(* Logix 5000 project; controller NorthLineDepalletizerPLC vendor 1 type 14 code 106 rev 33.11; software revision 33.00 *)

TASK MainTask (continuous, watchdog 500 ms) : MainProgram, Motoman, Comms

MODULES
   Local : vendor 1 type 14 code 106 (Compact 0, rev 33.11)
      BrazingOvenEthernetCard : 1756-ENBT (Ethernet 192.168.1.100, rev 5.1, Output RPI 10 ms)
         BrazingOvenPLC : vendor 1 type 14 code 92 (ICP 0, rev 24.1, $af6df9d4$ RPI 20 ms)
      cam : vendor 678 type 100 code 276 (Ethernet 192.168.1.33, rev 11.1, Output RPI 60 ms)
      YRC1000_Rbt_Ctlr : ETHERNET-MODULE (Ethernet 192.168.1.31, rev 1.1, Output RPI 10 ms)
      Fanuc_5 : ETHERNET-MODULE (Ethernet 192.168.1.5, rev 1.1, Output RPI 10 ms)
           Fanuc_5:I.Data[2]   // Part Count from Fanuc
           Fanuc_5:O.Data[0]   // Part Width to give to Fanuc
           Fanuc_5:O.Data[3]   // Part Length to give to Fanuc
           Fanuc_5:O.Data[1]   // Part ID to give to Fanuc
           Fanuc_5:O.Data[4]   // Part Count to give to Fanuc
           Fanuc_5:O.Data[2]   // Conveyor Height to pass along to Fanuc
      IFM_AL1322 : vendor 322 type 12 code 1322 (Ethernet 192.168.1.32, rev 1.6, StandardDataDriven RPI 10 ms)
END_MODULES

TYPE PatternResult :
STRUCT
   Angle : REAL;
   Score : REAL;
   X : REAL;
   Y : REAL;
END_STRUCT
END_TYPE

TYPE YRC1000_POSITION_VAR :
STRUCT
   Data_Type : DINT;   // Position Data Type of the Following Data 0: Pulse 16: Base 17: Robot 18: Tool 19: User coordinates
   Config : DINT;   // The configuration will be output bit 0: Back bit 1: Lower arm bit 2: No flip bit 3: R axis ≥ 180° bit 4: T axis ≥ 180° bit 5: S axis ≥ 180°
   Tool_Num : DINT;   // Tool #
   User_Coord_Num : DINT;   // User Coordinate #
   Ext_Config : DINT;   // Output the 7-axis robot extended configuration bit 0: θL ≥ 180° bit 1: θU ≥ 180° bit 2: θB ≥ 180° bit 3: θE ≥ 180° bit 4: θW ≥ 180°
   Axis1_Data : DINT;   // For pulse: Each axis’ pulse value For base: Length (μm) Angle (0.0001°)
   Axis2_Data : DINT;   // For pulse: Each axis’ pulse value For base: Length (μm) Angle (0.0001°)
   Axis3_Data : DINT;   // For pulse: Each axis’ pulse value For base: Length (μm) Angle (0.0001°)
   Axis4_Data : DINT;   // For pulse: Each axis’ pulse value For base: Length (μm) Angle (0.0001°)
   Axis5_Data : DINT;   // For pulse: Each axis’ pulse value For base: Length (μm) Angle (0.0001°)
   Axis6_Data : DINT;   // For pulse: Each axis’ pulse value For base: Length (μm) Angle (0.0001°)
   Axis7_Data : DINT;   // For pulse: Each axis’ pulse value For base: Length (μm) Angle (0.0001°)
   Axis8_Data : DINT;   // For pulse: Each axis’ pulse value For base: Length (μm) Angle (0.0001°)
END_STRUCT
END_TYPE

ADD_ON_INSTRUCTION Generic_8PORT_IOL   (* revision 3.0 *)
// Revision note:
// 12/2022:updated to current AOI standards:LH
VAR_IN_OUT
   PLC_Input : INT[223]; {required}   // Reference the Input Controller tag <IOLinkMasterName>:I1.Data
   PLC_Output : INT[151]; {required}   // Reference the Output Controller tag <IOLinkMasterName>:O1.Data
END_VAR
VAR_INPUT
   Port_Process_Data_Size : SINT := 4;   // User Input Value from the Configuration Controller tag <IOLinkMasterName>:C.Port_Process_Data_Size
   Port_Number : SINT; {visible}   // User Input Value = Port number of the IO-Link Master
END_VAR
VAR_OUTPUT
   Vendor_ID : INT; {access Read Only, visible}   // Read only value indicating the manufacturer of the IO-Link Device. ifm=310 dec
   Device_ID : DINT; {access Read Only, visible}   // Read only value set by the manufacturer of the device. Varies by product family
   IOL_Mode : BOOL; {access Read Only, visible}   // True: Port is configured for IO-Link Communication. False: Port is not configured for IO-Link Communication
   Device_Not_Connected : BOOL; {access Read Only, visible}   // True: No IO-Link Device is connected False: IO-Link Device is connected
   Invalid_Data : BOOL; {access Read Only, visible}   // True: IO-Link Data is invalid False: IO-Link Data is valid
   Wrong_VID_DID : BOOL; {access Read Only, visible}   // True: Vendor ID and/or Device ID does not match the configured VID or DID set in Configuration Controller Tag(s) <IOLink MasterName>:C.Vendor_ID_Port_n or ...C.Device_ID_Port_n
   Diagnostic_Avail : BOOL; {access Read Only, visible}   // True: IO-Link Event data is available False: No Event data is present
   AOI_Settings_Error : BOOL; {access Read Only, visible}   // A user input is out of range. Check port process data size and port number
END_VAR
VAR_IN_OUT
   Input_Data_Array : INT[16]; {required}   // Up to 16 words/32 bytes of Input process data produced by the IO-Link device
        [5]   // Input Word 5/Byte 10 0..7/Byte 11 8..15
        [0]   // Input Word 0/Byte 0 0..7/Byte 1 8..15
        [1]   // Input Word 1/Byte 2 0..7/Byte 3 8..15
        [6]   // Input Word 6/Byte 12 0..7/Byte 13 8..15
        [2]   // Input Word 2/Byte 4 0..7/Byte 5 8..15
        [7]   // Input Word 7/Byte 14 0..7/Byte 15 8..15
        [8]   // Input Word 8/Byte 16 0..7/Byte 17 8..15
        [9]   // Input Word 9/Byte 18 0..7/Byte 19 8..15
        [3]   // Input Word 3/Byte 6 0..7/Byte 7 8..15
        [10]   // Input Word 10/Byte 20 0..7/Byte 21 8..15
        [11]   // Input Word 11/Byte 22 0..7/Byte 23 8..15
        [12]   // Input Word 12/Byte 24 0..7/Byte 25 8..15
        [13]   // Input Word 13/Byte 26 0..7/Byte 27 8..15
        [14]   // Input Word 14/Byte 28 0..7/Byte 29 8..15
        [15]   // Input Word 15/Byte 30 0..7/Byte 31 8..15
        [4]   // Input Word 4/Byte 8 0..7/Byte 9 8..15
   Output_Data_Array : INT[16]; {required}   // Up to 32 bytes of Output process data consumed by the IO-Link device
        [0]   // Output Word 0/Byte 1 0..7/Byte 0 8..15
        [1]   // Output Word 1/Byte 3 0..7/Byte 2 8..15
        [5]   // Output Word 5/Byte 11 0..7/Byte 10 8..15
        [6]   // Output Word 6/Byte 13 0..7/Byte 12 8..15
        [7]   // Output Word 7/Byte 15 0..7/Byte 14 8..15
        [8]   // Output Word 8/Byte 17 0..7/Byte 16 8..15
        [9]   // Output Word 9/Byte 19 0..7/Byte 18 8..15
        [2]   // Output Word 2/Byte 5 0..7/Byte 4 8..15
        [3]   // Output Word 3/Byte 7 0..7/Byte 6 8..15
        [10]   // Output Word 10/Byte 21 0..7/Byte 20 8..15
        [4]   // Output Word 4/Byte 9 0..7/Byte 8 8..15
        [11]   // Output Word 11/Byte 23 0..7/Byte 22 8..15
        [12]   // Output Word 12/Byte 25 0..7/Byte 24 8..15
        [13]   // Output Word 13/Byte 27 0..7/Byte 26 8..15
        [14]   // Output Word 14/Byte 29 0..7/Byte 28 8..15
        [15]   // Output Word 15/Byte 31 0..7/Byte 30 8..15
END_VAR
VAR
   Data_Size : SINT; {access None}   // Factor of the RealPort_Num to calcualated the Offset_Address
   Offset_StatusFlgs : SINT; {access None}   // RealPort_Num+9
   RealPort_Num : SINT; {access None}   // Result of the Port_Number-1
   StatusFlgs_Offset : SINT; {access None}   // Result of Offset_StatusFlgs+23
   Offset_Address : INT; {access None}   // Result of Data_Size*RealPort_Number
   Process_Offset : INT; {access None}   // Result of Offset_Address+95(8port Master) or Offset_Address+59(4port Master). Used to indicate the word offset for where the IO-Link device’s process input data starts
   Process_Out_Offset : INT; {access None}   // Result of Offset_Address+23
END_VAR

ROUTINE Logic   (* ladder *)
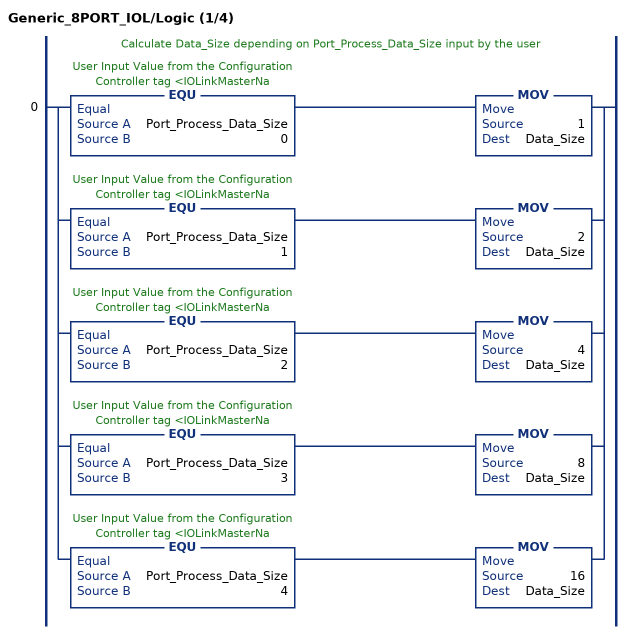
   // Calculate Data_Size depending on Port_Process_Data_Size input by the user
   0: [EQU(Port_Process_Data_Size,0) MOV(1,Data_Size) ,EQU(Port_Process_Data_Size,1) MOV(2,Data_Size) ,EQU(Port_Process_Data_Size,2) MOV(4,Data_Size) ,EQU(Port_Process_Data_Size,3) MOV(8,Data_Size) ,EQU(Port_Process_Data_Size,4) MOV(16,Data_Size) ];
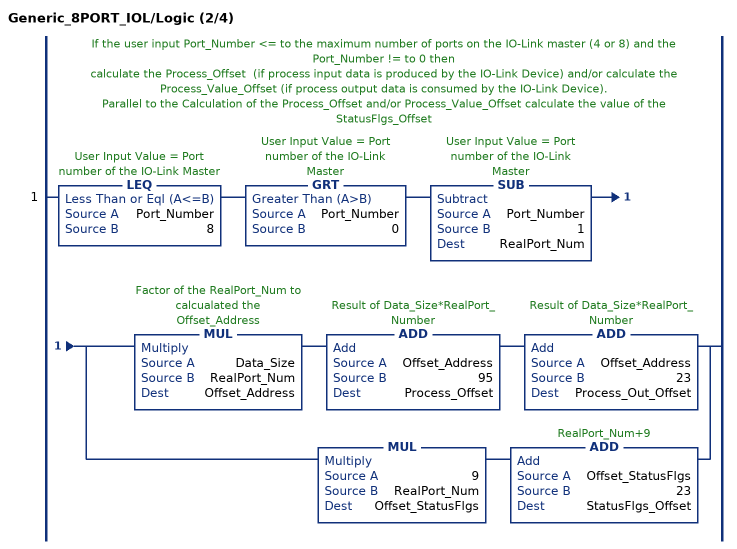
   // If the user input Port_Number <= to the maximum number of ports on the IO-Link master (4 or 8) and the Port_Number != to 0 then
   // calculate the Process_Offset  (if process input data is produced by the IO-Link Device) and/or calculate the Process_Value_Offset (if process output data is consumed by the IO-Link Device).
   // Parallel to the Calculation of the Process_Offset and/or Process_Value_Offset calculate the value of the StatusFlgs_Offset
   1: LEQ(Port_Number,8)GRT(Port_Number,0)SUB(Port_Number,1,RealPort_Num)[MUL(Data_Size,RealPort_Num,Offset_Address) ADD(Offset_Address,95,Process_Offset) ADD(Offset_Address,23,Process_Out_Offset) ,MUL(9,RealPort_Num,Offset_StatusFlgs) ADD(Offset_StatusFlgs,23,StatusFlgs_Offset) ];
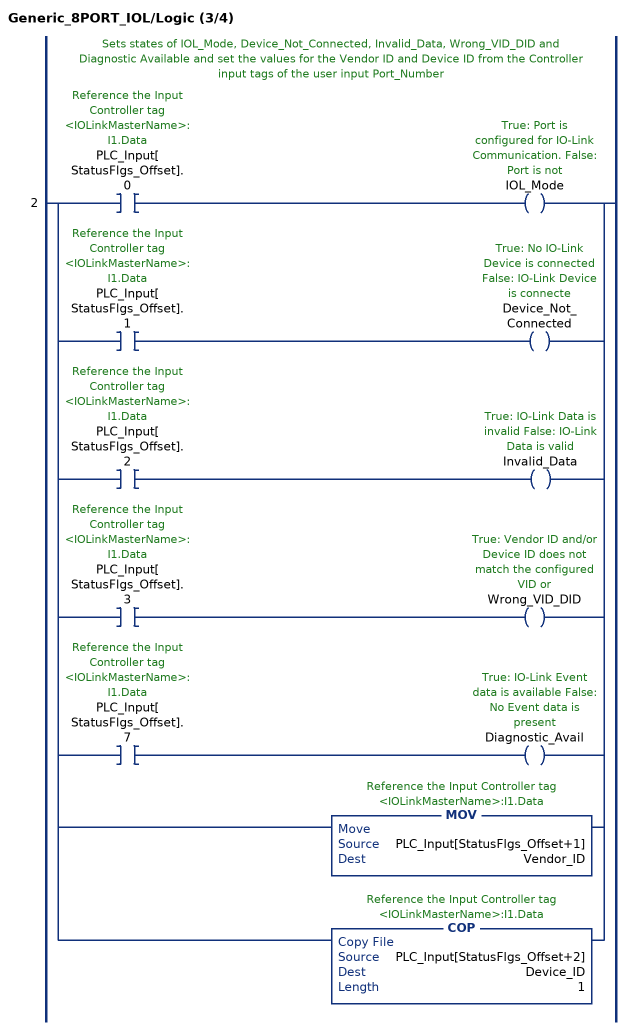
   // Sets states of IOL_Mode, Device_Not_Connected, Invalid_Data, Wrong_VID_DID and Diagnostic Available and set the values for the Vendor ID and Device ID from the Controller input tags of the user input Port_Number
   2: [XIC(PLC_Input[StatusFlgs_Offset].0) OTE(IOL_Mode) ,XIC(PLC_Input[StatusFlgs_Offset].1) OTE(Device_Not_Connected) ,XIC(PLC_Input[StatusFlgs_Offset].2) OTE(Invalid_Data) ,XIC(PLC_Input[StatusFlgs_Offset].3) OTE(Wrong_VID_DID) ,XIC(PLC_Input[StatusFlgs_Offset].7) OTE(Diagnostic_Avail) ,MOV(PLC_Input[StatusFlgs_Offset+1],Vendor_ID) ,COP(PLC_Input[StatusFlgs_Offset+2],Device_ID,1) ];
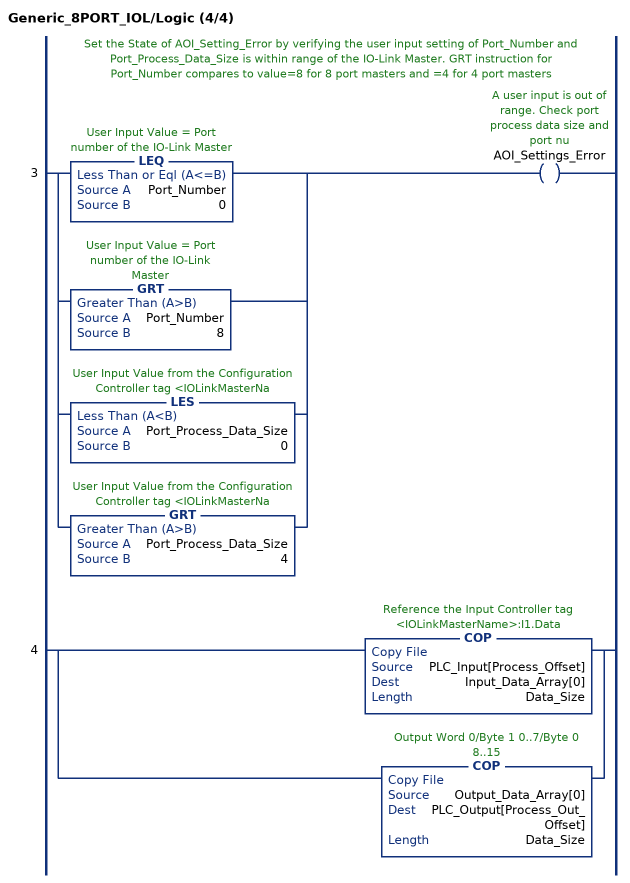
   // Set the State of AOI_Setting_Error by verifying the user input setting of Port_Number and Port_Process_Data_Size is within range of the IO-Link Master. GRT instruction for Port_Number compares to value=8 for 8 port masters and =4 for 4 port masters
   3: [LEQ(Port_Number,0) ,GRT(Port_Number,8) ,LES(Port_Process_Data_Size,0) ,GRT(Port_Process_Data_Size,4) ]OTE(AOI_Settings_Error);
   4: [COP(PLC_Input[Process_Offset],Input_Data_Array[0],Data_Size) ,COP(Output_Data_Array[0],PLC_Output[Process_Out_Offset],Data_Size) ];
END_ROUTINE
END_ADD_ON_INSTRUCTION

VAR_GLOBAL   (* controller tags *)
   AcknowledgeCameraImage : ALIAS FOR YRC1000_Rbt_Ctlr:O.Data[4].5;
   AcknowledgeHeightCheck : ALIAS FOR YRC1000_Rbt_Ctlr:O.Data[4].4;
   AcknowledgeLevelCheck : ALIAS FOR YRC1000_Rbt_Ctlr:O.Data[6].4;
   AcknowledgePalletTooTall : ALIAS FOR YRC1000_Rbt_Ctlr:O.Data[7].4;
   ActiveUserFrame : DINT;   // Currently Active Pallet
   AirPressure : ALIAS FOR YRC1000_Rbt_Ctlr:I.Data[1].4;
   Alarm : ALIAS FOR YRC1000_Rbt_Ctlr:I.Data[8].3;
   AlarmReset : ALIAS FOR YRC1000_Rbt_Ctlr:O.Data[0].3;
   AngleHeightCheck : ALIAS FOR YRC1000_Rbt_Ctlr:I.Data[10].4;
   AtHomePosition : ALIAS FOR YRC1000_Rbt_Ctlr:I.Data[5].2;
   BatteryAlarm : ALIAS FOR YRC1000_Rbt_Ctlr:I.Data[8].4;
   Blue1 : BOOL;
   Blue2 : BOOL;
   CallMaster : ALIAS FOR YRC1000_Rbt_Ctlr:O.Data[0].2;
   CameraAngle : REAL := 0.56835175;
   CameraFailed : ALIAS FOR YRC1000_Rbt_Ctlr:O.Data[5].7;
   CameraJobName : STRING := '2832_SingleStackACoils.job';
   CameraOffsetX : REAL := 0.8950585;
   CameraOffsetY : REAL := -5.923684;
   CameraScore : REAL := 1.0;
   CamJobData : SINT[32] := ([0] := 26, [2] := 50, [3] := 56, [4] := 51, [5] := 50, [6] := 95, [7] := 83, [8] := 105, [9] := 110, [10] := 103, [11] := 108, [12] := 101, [13] := 83, [14] := 116, [15] := 97, [16] := 99, [17] := 107, [18] := 65, [19] := 67, [20] := 111, [21] := 105, [22] := 108, [23] := 115, [24] := 46, [25] := 106, [26] := 111, [27] := 98);
   CapacitiveInArray : INT[16] := ([0] := 928);
   CapacitiveOutArray : INT[16];
   CapacitiveSensorValue : DINT := 58;
   ccr0 : DINT;
   ccr1 : DINT := 1;
   ccr2 : DINT := 2;
   ChangingJob : BOOL;
   CoilLocation : YRC1000_POSITION_VAR := (Data_Type := 19, Tool_Num := 2, User_Coord_Num := 5, Axis1_Data := 895, Axis2_Data := -5924, Axis3_Data := 15000, Axis4_Data := 1800000, Axis6_Data := -1794316);
   CoilLocationFound : ALIAS FOR YRC1000_Rbt_Ctlr:O.Data[4].6;
   CoilType : DINT := 1;   // 1: 17" 2: 30" 3: 41"
   CompleteState : DINT := 100;
   ConvertedCameraResults : REAL[3] := ([0] := 0.8950585, [1] := -5.923684, [2] := -179.43164);
   ConveyorApproach : YRC1000_POSITION_VAR := (Data_Type := 19, Tool_Num := 8, User_Coord_Num := 3, Axis2_Data := -50000, Axis3_Data := 151600, Axis4_Data := 1800000, Axis5_Data := 100000, Axis6_Data := -900000);
   ConveyorBeforePlace : YRC1000_POSITION_VAR := (Data_Type := 19, Tool_Num := 8, User_Coord_Num := 3, Axis2_Data := -10000, Axis3_Data := 56600, Axis4_Data := 1800000, Axis5_Data := 100000, Axis6_Data := -900000);
   ConveyorIn : YRC1000_POSITION_VAR := (Data_Type := 19, Tool_Num := 8, User_Coord_Num := 3, Axis2_Data := -50000, Axis3_Data := 56600, Axis4_Data := 1800000, Axis5_Data := 100000, Axis6_Data := -900000);
   ConveyorOver : YRC1000_POSITION_VAR := (Data_Type := 19, Tool_Num := 8, User_Coord_Num := 3, Axis2_Data := -50000, Axis3_Data := 151600, Axis4_Data := 1800000, Axis5_Data := 100000, Axis6_Data := -900000);
   Corner1Dist : DINT := 1499300;
   Corner2Dist : DINT := 1508800;
   Corner3Dist : DINT := 1504500;
   Corner4Dist : DINT := 1504900;
   Cos30 : REAL := 0.8660254;
   Cos45 : REAL := 0.70710677;
   CurrentPos : REAL[6] := ([0] := 1000.0, [2] := 799.997, [3] := 180.0, [4] := -0.0003, [5] := -1.e-04);   // Current position of the active TCP on the robot
   CurrentPosition_micro : YRC1000_POSITION_VAR := (Data_Type := 16, Config := 4, Tool_Num := 1, Axis1_Data := 1000000, Axis3_Data := 799997, Axis4_Data := 1800000, Axis5_Data := -3, Axis6_Data := -1);
   CurrentRobotTask : DINT := 5;
   delay_0017_Coil_Camera : TIMER := (PRE := 10);
   delay_0017_Orient_Camera : TIMER := (PRE := 10);
   delay_0017_PickLocation : TIMER := (PRE := 10, ACC := 10, EN := 1, DN := 1);
   delay_2832_Edge_Camera : TIMER := (PRE := 10);
   delay_2832_Edge_SearchLocation : TIMER := (PRE := 10);
   delay_2832_Middle_Camera : TIMER := (PRE := 10);
   delay_2832_Middle_SearchLocation : TIMER := (PRE := 10);
   delay_2832_PickLocation : TIMER := (PRE := 10);
   delay_3041_Edge_Camera : TIMER := (PRE := 10);
   delay_3041_Edge_SearchLocation : TIMER := (PRE := 10);
   delay_3041_Middle_Camera : TIMER := (PRE := 10);
   delay_3041_Middle_SearchLocation : TIMER := (PRE := 10, ACC := 11, EN := 1, DN := 1);
   delay_3041_PickLocation : TIMER := (PRE := 10, ACC := 11, EN := 1, DN := 1);
   delay_ActiveUserFrame : TIMER := (PRE := 10);
   delay_CurrentPos : TIMER := (PRE := 10);
   delay_LeftConveyorOff : TIMER := (PRE := 1000, ACC := 1000, EN := 1, DN := 1);
   delay_LeftConveyorOffLong : TIMER := (PRE := 60000);
   delay_LeftConveyorOn : TIMER := (PRE := 10);
   delay_LeftPalletOff : TIMER := (PRE := 1000);
   delay_LeftPalletOn : TIMER := (PRE := 1000, ACC := 1000, EN := 1, DN := 1);
   delay_PalletComplete : TIMER := (PRE := 10, ACC := 11, EN := 1, DN := 1);
   delay_Read_PartCount : TIMER := (PRE := 50, ACC := 4, EN := 1, TT := 1);
   delay_Read_RobotCurrentTask : TIMER := (PRE := 50, ACC := 38, EN := 1, TT := 1);
   delay_RightConveyorOff : TIMER := (PRE := 1000);
   delay_RightConveyorOffLong : TIMER := (PRE := 60000);
   delay_RightConveyorOn : TIMER := (PRE := 10, ACC := 10, EN := 1, DN := 1);
   delay_RightPalletOff : TIMER := (PRE := 1000, ACC := 1000, EN := 1, DN := 1);
   delay_RightPalletOn : TIMER := (PRE := 1000);
   DiffHeightCheckVal : DINT := 9500;   // Difference between the highest and shortest corners of a pallet
   DistanceInArray : INT[16] := ([0] := 22177);
        [0]   // Distance sensor reading in 0.1 mm
   DistanceOutArray : INT[16];
   DistanceSensorValue_micro : DINT := 2217600;
   DoorEntryRequested : ALIAS FOR YRC1000_Rbt_Ctlr:O.Data[5].3;
   DoorLatchRelayPower : ALIAS FOR YRC1000_Rbt_Ctlr:O.Data[2].3;
   DoorRequestAccess : ALIAS FOR YRC1000_Rbt_Ctlr:I.Data[1].0;
   DoorUnlocked : ALIAS FOR YRC1000_Rbt_Ctlr:I.Data[1].7;
   err_CameraFailed : BOOL;
   err_HeightCheckInconsistent : ALIAS FOR YRC1000_Rbt_Ctlr:O.Data[6].3;
   err_RobotPickupFailed : ALIAS FOR YRC1000_Rbt_Ctlr:I.Data[10].3;
   ErrorState : DINT := 99;
   ExternalHold : ALIAS FOR YRC1000_Rbt_Ctlr:O.Data[0].1;
   ExternalServoOn : ALIAS FOR YRC1000_Rbt_Ctlr:O.Data[0].4;
   ExternalStart : ALIAS FOR YRC1000_Rbt_Ctlr:O.Data[0].0;
   FailedCaptures : DINT;   // Number of times the camera failed to find the coil
   FanucLongPart : DINT := 1072;
   FanucMediumPart : DINT := 795;
   FanucShortPart : DINT := 465;
   FoundPattern : DINT;
   GoHome : ALIAS FOR YRC1000_Rbt_Ctlr:O.Data[6].6;
   GoodToPick : ALIAS FOR YRC1000_Rbt_Ctlr:O.Data[8].0;
   GoToToolChange : ALIAS FOR YRC1000_Rbt_Ctlr:O.Data[6].0;
   Green1 : BOOL;
   Green2 : BOOL;
   Gripper_Extend : ALIAS FOR YRC1000_Rbt_Ctlr:I.Data[10].0;
   Gripper_Extended : ALIAS FOR YRC1000_Rbt_Ctlr:O.Data[5].0;
   Gripper_HoldingPart : ALIAS FOR YRC1000_Rbt_Ctlr:O.Data[4].7;
   Gripper_Retract : ALIAS FOR YRC1000_Rbt_Ctlr:I.Data[10].1;
   Gripper_Retracted : ALIAS FOR YRC1000_Rbt_Ctlr:O.Data[5].1;
   HeightCheck1 : ALIAS FOR YRC1000_Rbt_Ctlr:I.Data[9].0;
   HeightCheck2 : ALIAS FOR YRC1000_Rbt_Ctlr:I.Data[9].1;
   HeightCheck3 : ALIAS FOR YRC1000_Rbt_Ctlr:I.Data[9].2;
   HeightCheck4 : ALIAS FOR YRC1000_Rbt_Ctlr:I.Data[9].3;
   HeightCheckAngled : REAL := 1886376.5;
   HeightCheckAvg : DINT := 1504375;
   HeightCheckTotal : DINT := 6017500;
   HighestCorner : DINT;   // Index of the highest corner on a quad-stack pallet
   HMI_GoHome : BOOL;
   HMI_Reset : BOOL;
   HMI_Start : BOOL;
   HMI_Stop : BOOL;
   HMI_Stop_Now : BOOL;
   HorizontalLineFound : BOOL;
   i : DINT := 3;
   IFM_Device_Disconnected : BOOL;
   InHomePosition : ALIAS FOR YRC1000_Rbt_Ctlr:O.Data[5].6;
   InPlay : ALIAS FOR YRC1000_Rbt_Ctlr:I.Data[8].6;
   InRemote : ALIAS FOR YRC1000_Rbt_Ctlr:I.Data[8].5;
   InTeach : ALIAS FOR YRC1000_Rbt_Ctlr:I.Data[8].7;
   InToolChange : ALIAS FOR YRC1000_Rbt_Ctlr:I.Data[10].5;
   j : DINT := 8;
   JobNamePrefix : STRING := '2832';
   JobResults : PatternResult[4] := ([0].Angle := 0.56835175, [0].Score := 1.0, [0].X := 0.8950585, [0].Y := -5.923684, [1].Angle := -0.24466617, [1].Score := 67.82552, [1].X := 22.508408, [1].Y := -36.919308, [2].Angle := -0.48321187, [2].Score := 95.65568, [2].X := -50.188633, [2].Y := 21.64503);   // Organized results from the most recent camera image
   LeftConveyorPresent : ALIAS FOR YRC1000_Rbt_Ctlr:O.Data[7].6;
   LeftConveyorSensor : ALIAS FOR YRC1000_Rbt_Ctlr:I.Data[1].5;
   LeftEdgeFound : ALIAS FOR YRC1000_Rbt_Ctlr:O.Data[6].7;
   LeftIndicator_Green : ALIAS FOR YRC1000_Rbt_Ctlr:O.Data[1].6;
   LeftIndicator_Yellow : ALIAS FOR YRC1000_Rbt_Ctlr:O.Data[1].7;
   LeftPalletComplete : ALIAS FOR YRC1000_Rbt_Ctlr:O.Data[4].0;
   LeftPalletPresent : ALIAS FOR YRC1000_Rbt_Ctlr:O.Data[7].1;
   LeftPalletSensor : ALIAS FOR YRC1000_Rbt_Ctlr:I.Data[1].2;
   LeftPalletWillBeNew : BOOL := 1;
   LevelCheck1 : ALIAS FOR YRC1000_Rbt_Ctlr:I.Data[10].7;
   LevelCheck2 : ALIAS FOR YRC1000_Rbt_Ctlr:I.Data[11].0;
   LevelCheck3 : ALIAS FOR YRC1000_Rbt_Ctlr:I.Data[11].1;
   LevelCheckBad : ALIAS FOR YRC1000_Rbt_Ctlr:O.Data[7].3;
   LevelCheckDone : ALIAS FOR YRC1000_Rbt_Ctlr:O.Data[6].5;
   LevelCheckStopPoint : DINT := 75;
   LoopsFound : BOOL;   // Used to determine if we are looking at the wrong end of a single-stack coil
   MaxHeightCheckVal : DINT := 1508800;
   MinHeightCheckVal : DINT := 1499300;
   msg_Read_ActiveUserFrame : MESSAGE;
        MessageParameters(ServiceCode := 16#000e, DestinationTag := ActiveUserFrame, ...)
   msg_Read_CurrentPosition : MESSAGE;
        MessageParameters(ServiceCode := 16#0001, DestinationTag := CurrentPosition_micro, ...)
   msg_Read_CurrentRobotTask : MESSAGE;
        MessageParameters(ServiceCode := 16#000e, DestinationTag := CurrentRobotTask, ...)
   msg_Read_PartCount : MESSAGE;
        MessageParameters(ServiceCode := 16#000e, DestinationTag := PartCount, ...)
   msg_Read_SearchLocation : MESSAGE;
        MessageParameters(ServiceCode := 16#000e, DestinationTag := SearchLocation, ...)
   msg_SetCamJob : MESSAGE; {access Read Only}
        MessageParameters(ServiceCode := 16#0010, LocalElement := CamJobData[0], ...)
   msg_Write_ActiveUserFrame : MESSAGE;
        MessageParameters(ServiceCode := 16#0010, LocalElement := ActiveUserFrame, ...)
   msg_Write_CoilLocation : MESSAGE;
        MessageParameters(ServiceCode := 16#0010, LocalElement := CoilLocation, ...)
   msg_Write_CoilType : MESSAGE;
        MessageParameters(ServiceCode := 16#0010, LocalElement := CoilType, ...)
   msg_Write_ConveyorApproach : MESSAGE;
        MessageParameters(ServiceCode := 16#0010, LocalElement := ConveyorApproach, ...)
   msg_Write_ConveyorBeforePlace : MESSAGE;
        MessageParameters(ServiceCode := 16#0010, LocalElement := ConveyorBeforePlace, ...)
   msg_Write_ConveyorIn : MESSAGE;
        MessageParameters(ServiceCode := 16#0010, LocalElement := ConveyorIn, ...)
   msg_Write_ConveyorOver : MESSAGE;
        MessageParameters(ServiceCode := 16#0010, LocalElement := ConveyorOver, ...)
   msg_Write_HeightCheckAverage : MESSAGE;
        MessageParameters(ServiceCode := 16#0010, LocalElement := HeightCheckAvg, ...)
   msg_Write_HighestCorner : MESSAGE;
        MessageParameters(ServiceCode := 16#0010, LocalElement := HighestCorner, ...)
   msg_Write_PartCount : MESSAGE;
        MessageParameters(ServiceCode := 16#0010, LocalElement := PartCount, ...)
   msg_Write_SearchLocation : MESSAGE;
        MessageParameters(ServiceCode := 16#0010, LocalElement := SearchLocation, ...)
   NewPallet : ALIAS FOR YRC1000_Rbt_Ctlr:O.Data[5].2;
   ons_AddPartToQueue : BOOL;
   ons_CallMaster : BOOL;
   ons_IncPickFailCount : BOOL;
   ons_LatchStart : BOOL;
   ons_RemovePartFromQueue : BOOL;
   ons_Reset_0017Coil : BOOL;
   ons_Reset_0017Orient : BOOL;
   ons_Reset_2832Edge : BOOL;
   ons_Reset_2832Middle : BOOL;
   ons_Reset_3041Edge : BOOL;
   ons_Reset_3041Middle : BOOL;
   ons_Reset_CI_0017Coil : BOOL;
   ons_Reset_CI_0017Orient : BOOL := 1;
   ons_Reset_CI_2832Edge : BOOL;
   ons_Reset_CI_2832Middle : BOOL := 1;
   ons_Reset_CI_3041Edge : BOOL;
   ons_Reset_CI_3041Middle : BOOL;
   ons_Reset_PC_HeightCheck : BOOL;
   ons_StartHeightCheck : BOOL;
   ons_StartJob0017 : BOOL;
   ons_StartJob2832 : BOOL;
   ons_StartJob3041 : BOOL;
   ons_StartLevelCheck : BOOL;
   p : DINT := 2;
   PalletStarted : ALIAS FOR YRC1000_Rbt_Ctlr:I.Data[10].2;
   PalletTooTall : ALIAS FOR YRC1000_Rbt_Ctlr:I.Data[9].6;
   PartCount : DINT;   // Number of coils the robot has placed on either conveyor
   PartID : DINT := 9;
   PartLength : DINT := 432;
   PartLength_Current : DINT := 432;   // 17" = 432 mm 30" = 762 mm 41" = 1041 mm
   PartNum : DINT := 5990233;
   PartNum_Current : DINT := 5990124;
   PartNumber : STRING := '5990233';
   PartNumber_Current : STRING := '5990124';
   PartRows : DINT := 3;
   PartRows_Current : DINT := 3;
   PartThickness : REAL := 51.6;
   PartThickness_Current : REAL := 51.6;   // 2r = 34.1 - 34.8 mm 3r = 51.1 - 51.8 mm 4r = 68.2 - 68.9 mm
   PartWidth : DINT := 813;
   PartWidth_Current : DINT := 813;   // 14" = 356 mm 16" = 406 mm 20" = 508 mm 22" = 559 mm 24" = 610 mm 28" = 711 mm 32" = 813 mm
   patternToPickup : REAL := 178.0;   // Distance from provided pick position to actual pick position on single-stack A-coils
   PCConnect : STRING := '1/11/2024 2:51:13 PM';   // Used by HMI to determine connectivity
   PickFailCount : COUNTER := (PRE := 3);
   PickFailedThreeTimes : ALIAS FOR YRC1000_Rbt_Ctlr:O.Data[7].5;
   PickupErrorAcknowledge : ALIAS FOR YRC1000_Rbt_Ctlr:O.Data[5].5;
   Port1_Distance : Generic_8PORT_IOL := (Port_Process_Data_Size := 4, Port_Number := 1, Vendor_ID := 26, Device_ID := 6488065, IOL_Mode := 1);
   Port2_Stroke : Generic_8PORT_IOL := (Port_Process_Data_Size := 4, Port_Number := 2, Vendor_ID := 26, Device_ID := 8388785, IOL_Mode := 1);
   Port5_Capacitive : Generic_8PORT_IOL := (Port_Process_Data_Size := 4, Port_Number := 5, Vendor_ID := 310, Device_ID := 388, IOL_Mode := 1);
   QuadStack : ALIAS FOR YRC1000_Rbt_Ctlr:O.Data[4].3;
   QuadStackConfiguration1 : ALIAS FOR YRC1000_Rbt_Ctlr:O.Data[6].1;
   QuadStackConfiguration2 : ALIAS FOR YRC1000_Rbt_Ctlr:O.Data[6].2;
   Queue_PartCount : DINT[4];   // Queue of Part Counts to help keep track of what part info the Fanuc needs
   Queue_PartID : DINT[4] := ([0] := 9);   // Queue of Part IDs to send to the Fanuc
   Queue_PartLength : DINT[4] := ([0] := 432);   // Queue of Part Lengths to send to the Fanuc
   Queue_PartWidth : DINT[4] := ([0] := 813);   // Queue of Part Widths to send to the Fanuc
   Read_ActiveUserFrame : BOOL := 1;
   Read_CurrentPosition : BOOL := 1;
   Read_CurrentRobotTask : BOOL;
   Read_PartCount : BOOL;
   Read_SearchLocation : BOOL;
   recovery_CameraFailed : BOOL;
   recovery_HeightCheckFailed : BOOL;
   recovery_PalletTooTall : BOOL;
   recovery_PickupFailed : BOOL;
   Reset : ALIAS FOR YRC1000_Rbt_Ctlr:I.Data[1].1;
   RightConveyorPresent : ALIAS FOR YRC1000_Rbt_Ctlr:O.Data[7].7;
   RightConveyorSensor : ALIAS FOR YRC1000_Rbt_Ctlr:I.Data[1].6;
   RightEdgeFound : ALIAS FOR YRC1000_Rbt_Ctlr:O.Data[7].0;
   RightIndicator_Green : ALIAS FOR YRC1000_Rbt_Ctlr:O.Data[2].0;
   RightIndicator_Yellow : ALIAS FOR YRC1000_Rbt_Ctlr:O.Data[2].1;
   RightPalletComplete : ALIAS FOR YRC1000_Rbt_Ctlr:O.Data[4].1;
   RightPalletPresent : ALIAS FOR YRC1000_Rbt_Ctlr:O.Data[7].2;
   RightPalletSensor : ALIAS FOR YRC1000_Rbt_Ctlr:I.Data[1].3;
   RightPalletWillBeNew : BOOL := 1;
   RobotCameraRequest : ALIAS FOR YRC1000_Rbt_Ctlr:I.Data[9].4;
   RobotCurrentPalletComplete : ALIAS FOR YRC1000_Rbt_Ctlr:I.Data[10].6;
   RobotExternalEStop : ALIAS FOR YRC1000_Rbt_Ctlr:I.Data[4].1;
   RobotRequestStop : ALIAS FOR YRC1000_Rbt_Ctlr:O.Data[5].4;
   RobotTeachPendantEStop : ALIAS FOR YRC1000_Rbt_Ctlr:I.Data[4].2;
   RobotWentHome : ALIAS FOR YRC1000_Rbt_Ctlr:I.Data[9].5;
   run_0017_CE : BOOL;
   run_2832_CE : BOOL;
   run_3041_CE : BOOL;
   Running : ALIAS FOR YRC1000_Rbt_Ctlr:I.Data[8].0;
   RunPalletComplete : BOOL;
   SafetyCircuitBroken : ALIAS FOR YRC1000_Rbt_Ctlr:I.Data[4].0;
   SafetyConfig1 : ALIAS FOR YRC1000_Rbt_Ctlr:O.Data[2].5;
   SafetyConfig2 : ALIAS FOR YRC1000_Rbt_Ctlr:O.Data[2].6;
   SafetyConfig3 : ALIAS FOR YRC1000_Rbt_Ctlr:O.Data[2].7;
   SafetyRelayReset : ALIAS FOR YRC1000_Rbt_Ctlr:O.Data[2].4;
   SearchLocation : DINT := 3;   // Index of what part of the pallet the camera is looking at
   SelectedJobID : DINT := 2832;
   SelectPlay : ALIAS FOR YRC1000_Rbt_Ctlr:O.Data[0].5;
   SelectTeach : ALIAS FOR YRC1000_Rbt_Ctlr:O.Data[0].6;
   ServoOn : ALIAS FOR YRC1000_Rbt_Ctlr:I.Data[8].1;
   SingleStack : ALIAS FOR YRC1000_Rbt_Ctlr:O.Data[4].2;
   StackLight_Blue : ALIAS FOR YRC1000_Rbt_Ctlr:O.Data[1].3;
   StackLight_Buzzer : ALIAS FOR YRC1000_Rbt_Ctlr:O.Data[1].0;
   StackLight_Green : ALIAS FOR YRC1000_Rbt_Ctlr:O.Data[1].5;
   StackLight_Red : ALIAS FOR YRC1000_Rbt_Ctlr:O.Data[1].2;
   StackLight_White : ALIAS FOR YRC1000_Rbt_Ctlr:O.Data[1].1;
   StackLight_Yellow : ALIAS FOR YRC1000_Rbt_Ctlr:O.Data[1].4;
   state_CaptureImage : DINT := 100;
   state_ChangeJob : DINT := 100;
   state_HeightCheck : DINT := 100;
   state_Job0017 : DINT := 100;
   state_Job0017_Coil : DINT := 100;
   state_Job0017_Orient : DINT := 100;
   state_Job2832 : DINT;
   state_Job2832_Edge : DINT := 100;
   state_Job2832_Middle : DINT := 100;
   state_Job3041 : DINT;
   state_Job3041_Edge : DINT := 100;
   state_Job3041_Middle : DINT := 100;
   state_LevelCheck : DINT := 100;
   state_PalletComplete : DINT := 100;
   StrokeInputArray : INT[16] := ([0] := 12864);
   StrokeOutputArray : INT[16];
   StrokePosition : DINT := 804;   // Gripper Cylinder position GTE 700 = Retracted LTE 100 = Extended
   StuffingConveyorHeight : DINT := 1059;
   Test_FanucGrabbedAllParts : BOOL;
   timer_CallMaster : TIMER := (PRE := 5000);
   timer_GreenFlashOff : TIMER := (PRE := 1000);
   timer_GreenFlashOn : TIMER := (PRE := 1000);
   timer_HMI_Reset : TIMER := (PRE := 5000);
   timer_HMI_Start : TIMER := (PRE := 5000);
   timer_HMI_Stop : TIMER := (PRE := 500);
   timer_HoldingPart : TIMER := (PRE := 1000);
   timer_Job0017_CameraError : TIMER := (PRE := 30000);
   timer_Job2832_CameraError : TIMER := (PRE := 30000);
   timer_Job3041_CameraError : TIMER := (PRE := 30000);
   timer_LeftFlashOff : TIMER := (PRE := 1000);
   timer_LeftFlashOn : TIMER := (PRE := 1000);
   timer_ResultsValid : TIMER := (PRE := 5000);
   timer_RightFlashOff : TIMER := (PRE := 1000);
   timer_RightFlashOn : TIMER := (PRE := 1000);
   timer_SetCamJob : TIMER := (PRE := 5000);
   ToPC_ActivePallet : DINT;
   ToPC_AirPressure : DINT := 1;
   ToPC_CameraFailed : DINT;
   ToPC_CellStatus : DINT := 3;
   ToPC_DoorStatus : DINT := 2;
   ToPC_HeightCheckFailed : DINT;
   TOPC_IFMDeviceDisconnected : DINT;
   ToPC_InRemote : DINT;
   ToPC_LeftConveyorSensor : DINT;
   ToPC_LeftPalletStatus : DINT := 1;
   ToPC_PalletTooTall : DINT;
   ToPC_PickupFailed : DINT;
   ToPC_RightConveyorSensor : DINT := 1;
   ToPC_RightPalletStatus : DINT;
   ToPC_RobotAlarm : DINT;
   ToPC_RobotEStop : DINT := 1;
   ToPC_RobotRunning : DINT;
   ToPC_RobotSafetyStop : DINT := 1;
   ToPC_ToolStatus : DINT;
   TopOfMaster : ALIAS FOR YRC1000_Rbt_Ctlr:I.Data[8].2;
   VerticalLineFound : BOOL := 1;
   Write_ActiveUserFrame : BOOL;
   write_ActiveUserFrame_L : BOOL;
   Write_ActiveUserFrame_R : BOOL;
   Write_CoilLocation : BOOL;
   Write_CoilType : BOOL;
   Write_ConveyorPositions : BOOL;
   Write_HeightCheckAverage : BOOL;
   write_HighestCorner : BOOL;
   Write_PartCount : BOOL;
   Write_SearchLocation : BOOL;
END_VAR

PROGRAM Comms   (* main routine Main *)

ROUTINE Main   (* ladder *)
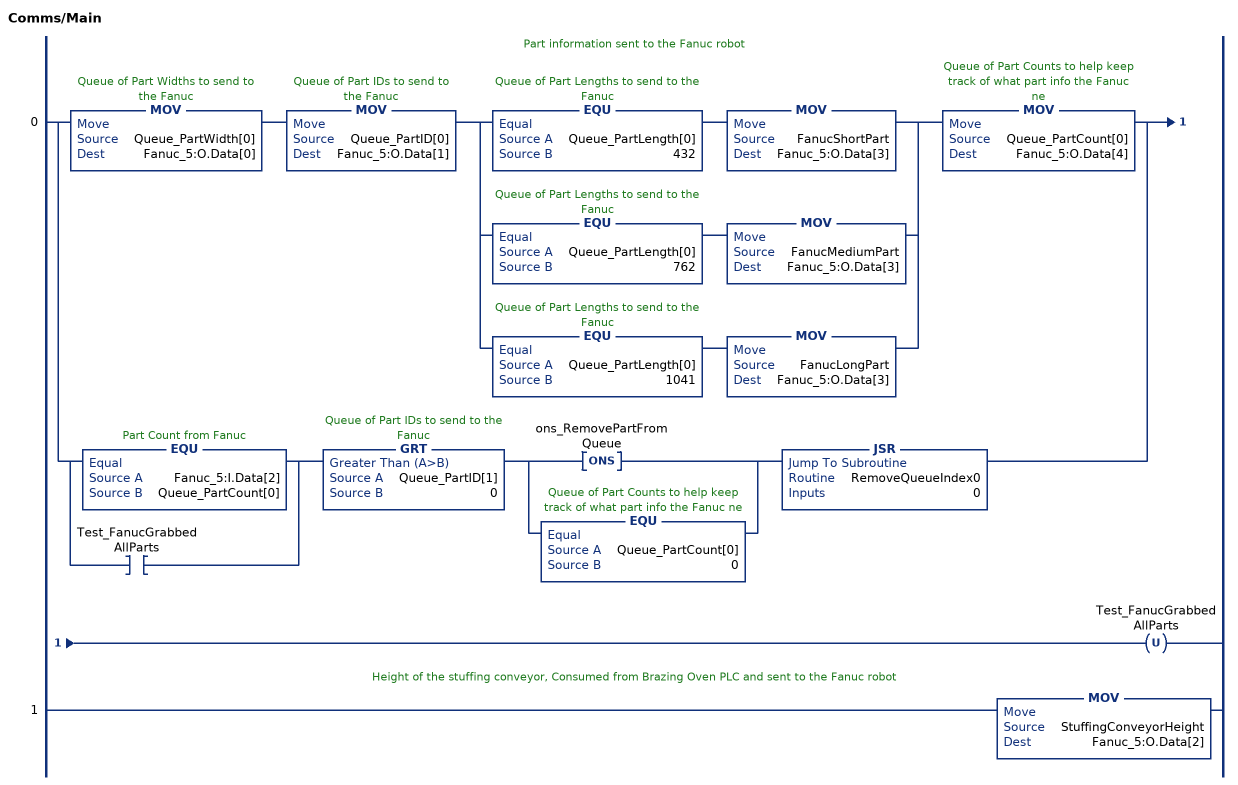
   // Part information sent to the Fanuc robot
   0: [MOV(Queue_PartWidth[0],Fanuc_5:O.Data[0]) MOV(Queue_PartID[0],Fanuc_5:O.Data[1]) [EQU(Queue_PartLength[0],432) MOV(FanucShortPart,Fanuc_5:O.Data[3]) ,EQU(Queue_PartLength[0],762) MOV(FanucMediumPart,Fanuc_5:O.Data[3]) ,EQU(Queue_PartLength[0],1041) MOV(FanucLongPart,Fanuc_5:O.Data[3]) ] MOV(Queue_PartCount[0],Fanuc_5:O.Data[4]) ,[EQU(Fanuc_5:I.Data[2],Queue_PartCount[0]) ,XIC(Test_FanucGrabbedAllParts) ] GRT(Queue_PartID[1],0) [ONS(ons_RemovePartFromQueue) ,EQU(Queue_PartCount[0],0) ] JSR(RemoveQueueIndex0,0) ]OTU(Test_FanucGrabbedAllParts);
   // Height of the stuffing conveyor, Consumed from Brazing Oven PLC and sent to the Fanuc robot
   1: MOV(StuffingConveyorHeight,Fanuc_5:O.Data[2]);
END_ROUTINE

ROUTINE RemoveQueueIndex0   (* structured text *)
   for i := 0 to 2 do
   	Queue_PartID[i] := Queue_PartID[i+1];
   end_for;
   Queue_PartID[3] := 0;
   
   for i := 0 to 2 do
   	Queue_PartCount[i] := Queue_PartCount[i+1];
   end_for;
   Queue_PartCount[3] := 0;
   
   for i := 0 to 2 do
   	Queue_PartLength[i] := Queue_PartLength[i+1];
   end_for;
   Queue_PartLength[3] := 0;
   
   for i := 0 to 2 do
   	Queue_PartWidth[i] := Queue_PartWidth[i+1];
   end_for;
   Queue_PartWidth[3] := 0;
END_ROUTINE
END_PROGRAM

PROGRAM MainProgram   (* main routine Main *)

ROUTINE CaptureImage   (* ladder *)
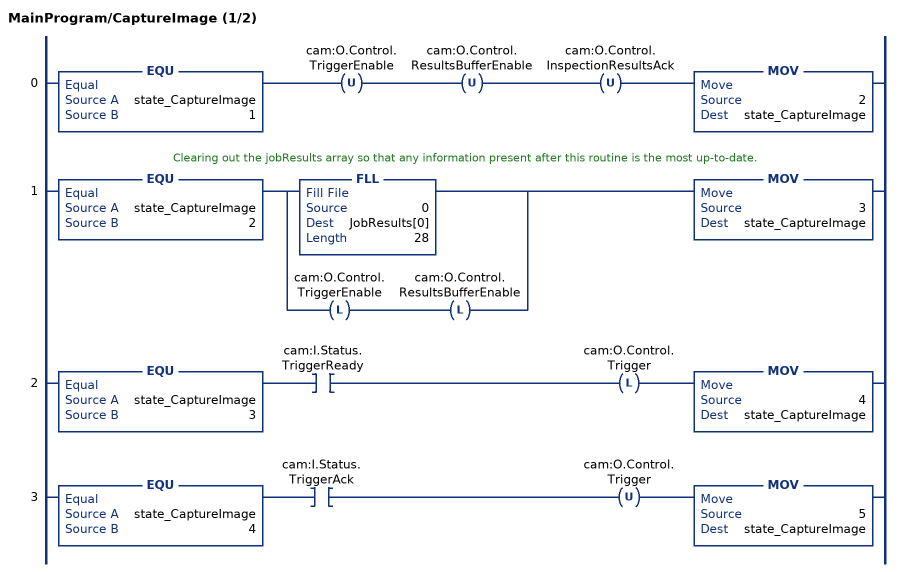
   0: EQU(state_CaptureImage,1)OTU(cam:O.Control.TriggerEnable)OTU(cam:O.Control.ResultsBufferEnable)OTU(cam:O.Control.InspectionResultsAck)MOV(2,state_CaptureImage);
   // Clearing out the jobResults array so that any information present after this routine is the most up-to-date.
   1: EQU(state_CaptureImage,2)[FLL(0,JobResults[0],28) ,OTL(cam:O.Control.TriggerEnable) OTL(cam:O.Control.ResultsBufferEnable) ]MOV(3,state_CaptureImage);
   2: EQU(state_CaptureImage,3)XIC(cam:I.Status.TriggerReady)OTL(cam:O.Control.Trigger)MOV(4,state_CaptureImage);
   3: EQU(state_CaptureImage,4)XIC(cam:I.Status.TriggerAck)OTU(cam:O.Control.Trigger)MOV(5,state_CaptureImage);
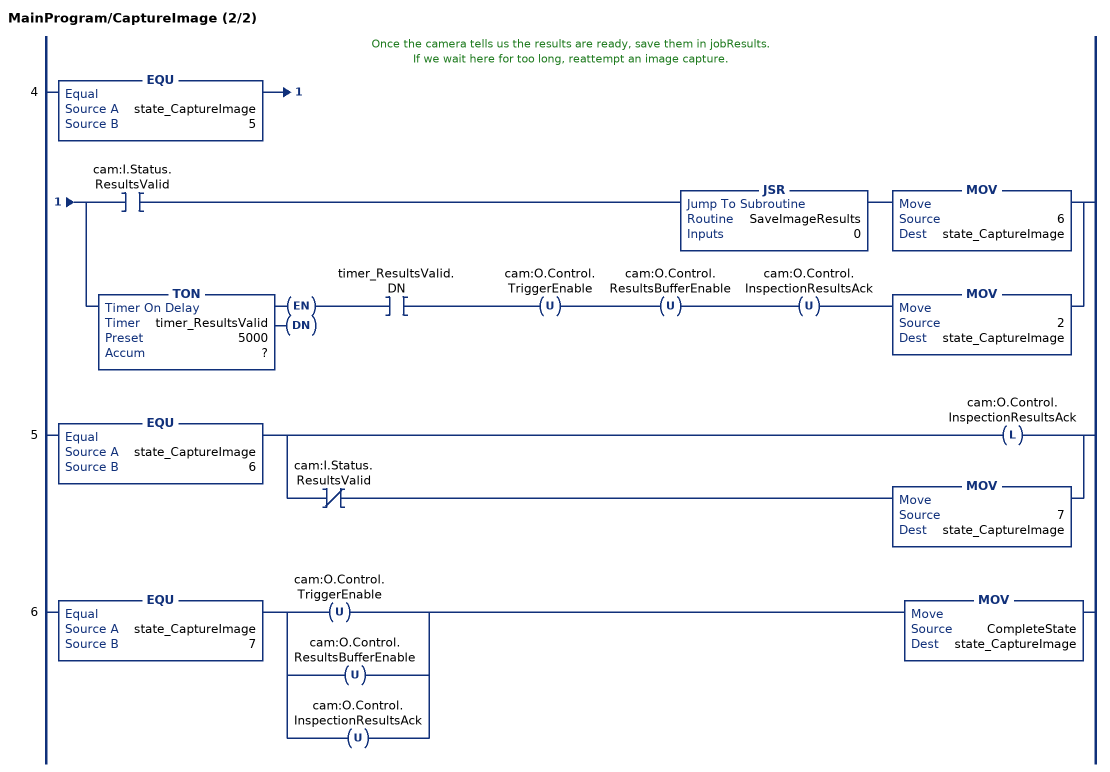
   // Once the camera tells us the results are ready, save them in jobResults.
   // If we wait here for too long, reattempt an image capture.
   4: EQU(state_CaptureImage,5)[XIC(cam:I.Status.ResultsValid) JSR(SaveImageResults,0) MOV(6,state_CaptureImage) ,TON(timer_ResultsValid,?,?) XIC(timer_ResultsValid.DN) OTU(cam:O.Control.TriggerEnable) OTU(cam:O.Control.ResultsBufferEnable) OTU(cam:O.Control.InspectionResultsAck) MOV(2,state_CaptureImage) ];
   5: EQU(state_CaptureImage,6)[OTL(cam:O.Control.InspectionResultsAck) ,XIO(cam:I.Status.ResultsValid) MOV(7,state_CaptureImage) ];
   6: EQU(state_CaptureImage,7)[OTU(cam:O.Control.TriggerEnable) ,OTU(cam:O.Control.ResultsBufferEnable) ,OTU(cam:O.Control.InspectionResultsAck) ]MOV(CompleteState,state_CaptureImage);
END_ROUTINE

ROUTINE ChangeCameraJob   (* ladder *)
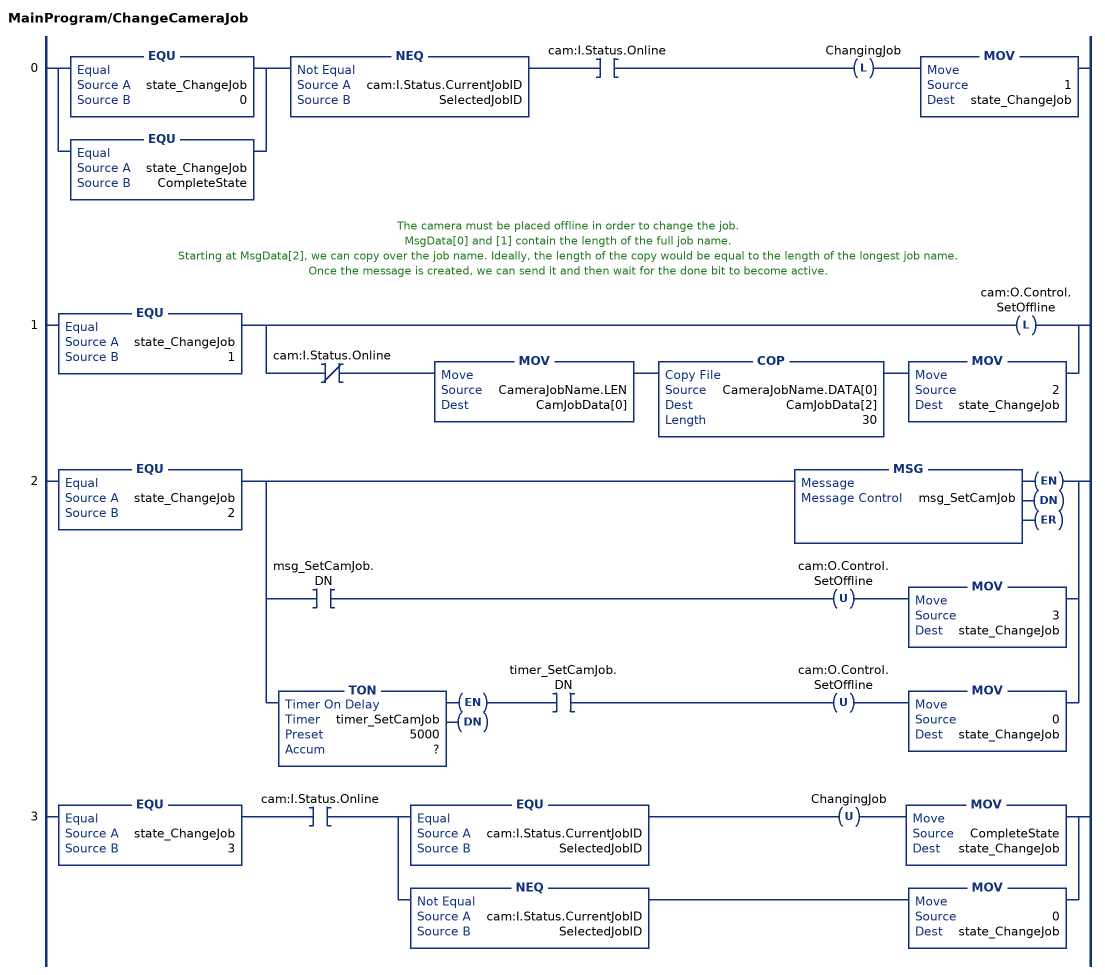
   0: [EQU(state_ChangeJob,0) ,EQU(state_ChangeJob,CompleteState) ]NEQ(cam:I.Status.CurrentJobID,SelectedJobID)XIC(cam:I.Status.Online)OTL(ChangingJob)MOV(1,state_ChangeJob);
   // The camera must be placed offline in order to change the job.
   // MsgData[0] and [1] contain the length of the full job name.
   // Starting at MsgData[2], we can copy over the job name. Ideally, the length of the copy would be equal to the length of the longest job name.
   // Once the message is created, we can send it and then wait for the done bit to become active.
   1: EQU(state_ChangeJob,1)[OTL(cam:O.Control.SetOffline) ,XIO(cam:I.Status.Online) MOV(CameraJobName.LEN,CamJobData[0]) COP(CameraJobName.DATA[0],CamJobData[2],30) MOV(2,state_ChangeJob) ];
   2: EQU(state_ChangeJob,2)[[MSG(msg_SetCamJob) ,XIC(msg_SetCamJob.DN) OTU(cam:O.Control.SetOffline) MOV(3,state_ChangeJob) ] ,TON(timer_SetCamJob,?,?) XIC(timer_SetCamJob.DN) OTU(cam:O.Control.SetOffline) MOV(0,state_ChangeJob) ];
   3: EQU(state_ChangeJob,3)XIC(cam:I.Status.Online)[EQU(cam:I.Status.CurrentJobID,SelectedJobID) OTU(ChangingJob) MOV(CompleteState,state_ChangeJob) ,NEQ(cam:I.Status.CurrentJobID,SelectedJobID) MOV(0,state_ChangeJob) ];
END_ROUTINE

ROUTINE CoilLocationData   (* structured text *)
   /*
   	This routine uses the values received from the camera
   	to set a position variable for the robot.
   */
   
   // Tool Number
   if PartLength_Current = 432 then
   	CoilLocation.Tool_Num := 2;
   elsif PartLength_Current = 762 then
   	CoilLocation.Tool_Num := 3;
   elsif PartLength_Current = 1041 then
   	CoilLocation.Tool_Num := 4;
   end_if;
   
   // X, Y, and Rz respectively
   CoilLocation.Axis1_Data := ConvertedCameraResults[ccr0] * 1000;
   CoilLocation.Axis2_Data := ConvertedCameraResults[ccr1] * 1000;
   CoilLocation.Axis3_Data := 15000;
   CoilLocation.Axis4_Data := 1800000;
   CoilLocation.Axis5_Data := 0;
   CoilLocation.Axis6_Data := ConvertedCameraResults[ccr2] * 10000;
END_ROUTINE

ROUTINE InterpretResults_0017   (* structured text *)
   /*
   	For this job, we only care about jobResults[0], which should be the pick position of the coil
   */
   
   if JobResults[0].Score > 0 then
   	FoundPattern := 0;
   
   	ConvertedCameraResults[0] := JobResults[0].X;
   	ConvertedCameraResults[1] := JobResults[0].Y;
   
   	if JobResults[0].Angle > 0 then
   		ConvertedCameraResults[2] := JobResults[0].Angle - 180;
   	else
   		ConvertedCameraResults[2] := JobResults[0].Angle + 180;
   	end_if;
   elsif JobResults[0].Score = 0 then
   	FoundPattern := -1;
   	RET();
   end_if;
END_ROUTINE

ROUTINE InterpretResults_2832   (* structured text *)
   /*
   	For this job, we only care about jobResults[0], which should be the pattern that we can offset from
   		to find our pick position.
   */
   
   if JobResults[0].Score > 0 then
   	FoundPattern := 0;
   
   	ConvertedCameraResults[0] := JobResults[FoundPattern].X + (patternToPickup * -SIN(RAD(JobResults[FoundPattern].Angle + 180)));
   	ConvertedCameraResults[1] := JobResults[FoundPattern].Y + (patternToPickup * COS(RAD(JobResults[FoundPattern].Angle + 180)));
   
   	if JobResults[FoundPattern].Angle > 0 then
   		ConvertedCameraResults[2] := JobResults[FoundPattern].Angle - 180;
   	else
   		ConvertedCameraResults[2] := JobResults[FoundPattern].Angle + 180;
   	end_if;
   elsif JobResults[0].Score = 0 then
   	FoundPattern := -1;
   	RET();
   end_if;
END_ROUTINE

ROUTINE InterpretResults_3041   (* structured text *)
   /*
   	For this job, we only care about jobResults[0], which should be the pick position of the coil
   */
   
   if JobResults[0].Score > 0 then
   	FoundPattern := 0;
   
   	ConvertedCameraResults[0] := JobResults[0].X;
   	ConvertedCameraResults[1] := JobResults[0].Y;
   
   	if JobResults[0].Angle > 0 then
   		ConvertedCameraResults[2] := JobResults[0].Angle - 180;
   	else
   		ConvertedCameraResults[2] := JobResults[0].Angle + 180;
   	end_if;
   elsif JobResults[0].Score = 0 then
   	FoundPattern := -1;
   	RET();
   end_if;
END_ROUTINE

ROUTINE InterpretResults_Middle   (* structured text *)
   /*
   	For this job, we only care about jobResults[1] and [2].
   		1 is a Vertical Line in the middle
   		2 is a Horizontal Line in the middle
   */
   
   // Reset these at the start
   VerticalLineFound := 0;
   HorizontalLineFound := 0;
   FoundPattern := -1;
   
   if JobResults[1].Score > 0 then
   	VerticalLineFound := 1;
   end_if;
   if JobResults[2].Score > 0 then
   	HorizontalLineFound := 1;
   end_if;
END_ROUTINE

ROUTINE IOLink   (* ladder *)
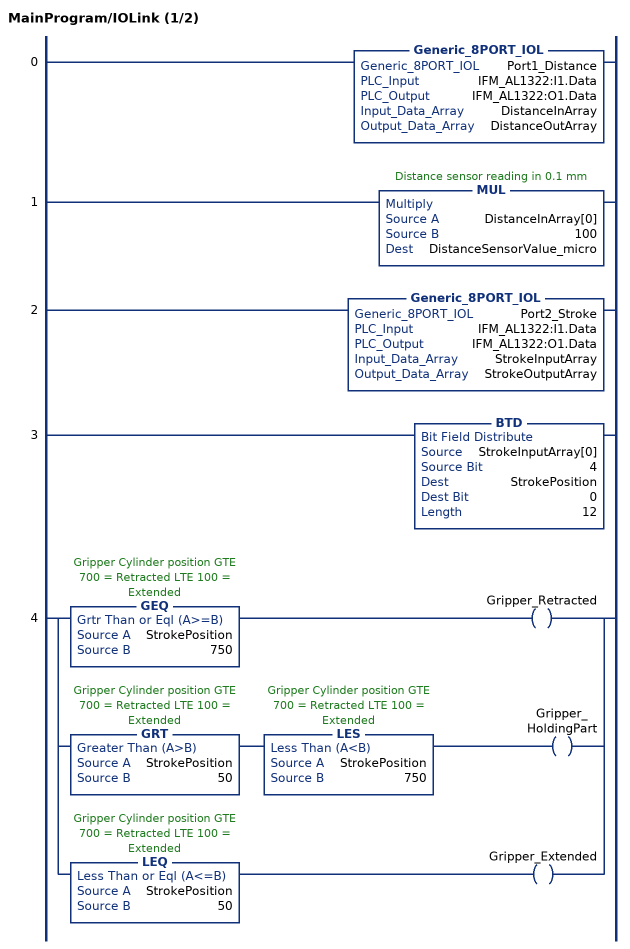
   0: Generic_8PORT_IOL(Port1_Distance,IFM_AL1322:I1.Data,IFM_AL1322:O1.Data,DistanceInArray,DistanceOutArray);
   1: MUL(DistanceInArray[0],100,DistanceSensorValue_micro);
   2: Generic_8PORT_IOL(Port2_Stroke,IFM_AL1322:I1.Data,IFM_AL1322:O1.Data,StrokeInputArray,StrokeOutputArray);
   3: BTD(StrokeInputArray[0],4,StrokePosition,0,12);
   4: [GEQ(StrokePosition,750) OTE(Gripper_Retracted) ,GRT(StrokePosition,50) LES(StrokePosition,750) OTE(Gripper_HoldingPart) ,LEQ(StrokePosition,50) OTE(Gripper_Extended) ];
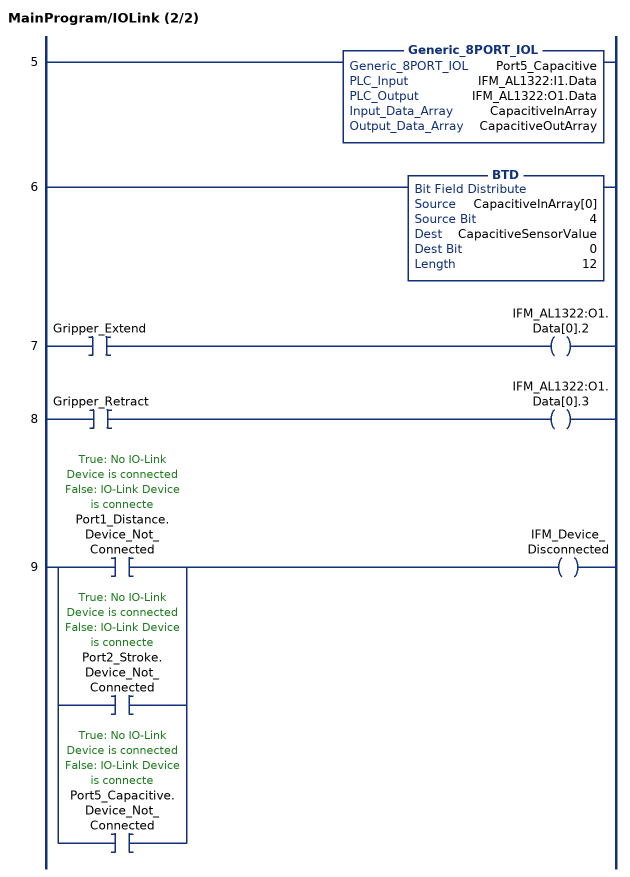
   5: Generic_8PORT_IOL(Port5_Capacitive,IFM_AL1322:I1.Data,IFM_AL1322:O1.Data,CapacitiveInArray,CapacitiveOutArray);
   6: BTD(CapacitiveInArray[0],4,CapacitiveSensorValue,0,12);
   7: XIC(Gripper_Extend)OTE(IFM_AL1322:O1.Data[0].2);
   8: XIC(Gripper_Retract)OTE(IFM_AL1322:O1.Data[0].3);
   9: [XIC(Port1_Distance.Device_Not_Connected) ,XIC(Port2_Stroke.Device_Not_Connected) ,XIC(Port5_Capacitive.Device_Not_Connected) ]OTE(IFM_Device_Disconnected);
END_ROUTINE

ROUTINE Job0017   (* ladder *)
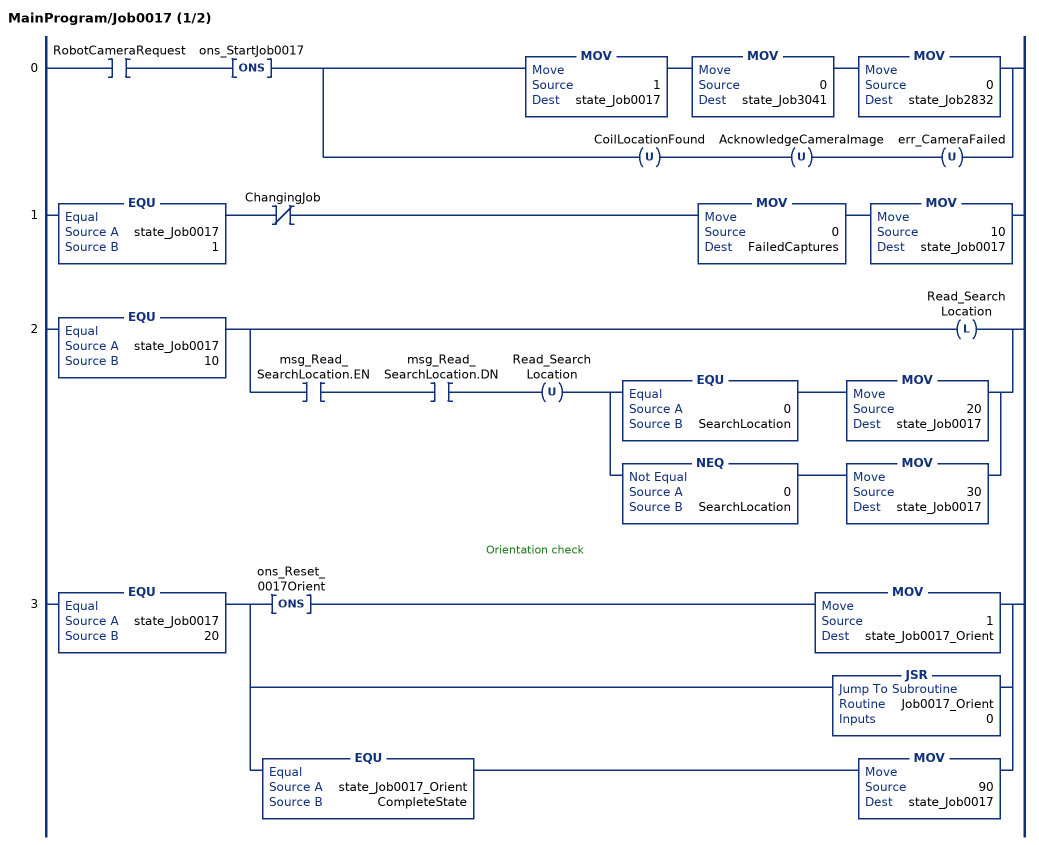
   0: XIC(RobotCameraRequest)ONS(ons_StartJob0017)[MOV(1,state_Job0017) MOV(0,state_Job3041) MOV(0,state_Job2832) ,OTU(CoilLocationFound) OTU(AcknowledgeCameraImage) OTU(err_CameraFailed) ];
   1: EQU(state_Job0017,1)XIO(ChangingJob)MOV(0,FailedCaptures)MOV(10,state_Job0017);
   2: EQU(state_Job0017,10)[OTL(Read_SearchLocation) ,XIC(msg_Read_SearchLocation.EN) XIC(msg_Read_SearchLocation.DN) OTU(Read_SearchLocation) [EQU(0,SearchLocation) MOV(20,state_Job0017) ,NEQ(0,SearchLocation) MOV(30,state_Job0017) ] ];
   // Orientation check
   3: EQU(state_Job0017,20)[[ONS(ons_Reset_0017Orient) MOV(1,state_Job0017_Orient) ,JSR(Job0017_Orient,0) ] ,EQU(state_Job0017_Orient,CompleteState) MOV(90,state_Job0017) ];
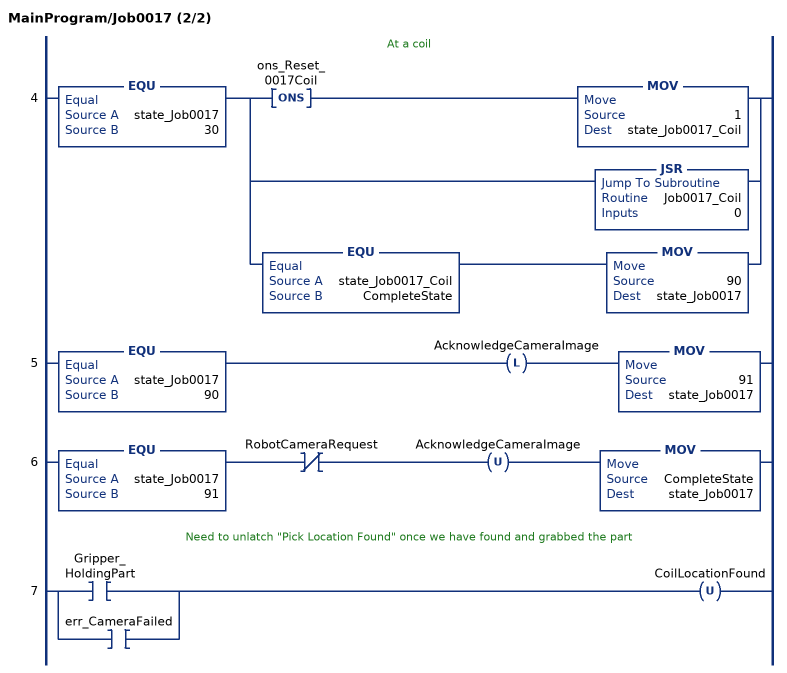
   // At a coil
   4: EQU(state_Job0017,30)[[ONS(ons_Reset_0017Coil) MOV(1,state_Job0017_Coil) ,JSR(Job0017_Coil,0) ] ,EQU(state_Job0017_Coil,CompleteState) MOV(90,state_Job0017) ];
   5: EQU(state_Job0017,90)OTL(AcknowledgeCameraImage)MOV(91,state_Job0017);
   6: EQU(state_Job0017,91)XIO(RobotCameraRequest)OTU(AcknowledgeCameraImage)MOV(CompleteState,state_Job0017);
   // Need to unlatch "Pick Location Found" once we have found and grabbed the part
   7: [XIC(Gripper_HoldingPart) ,XIC(err_CameraFailed) ]OTU(CoilLocationFound);
END_ROUTINE

ROUTINE Job0017_Coil   (* ladder *)
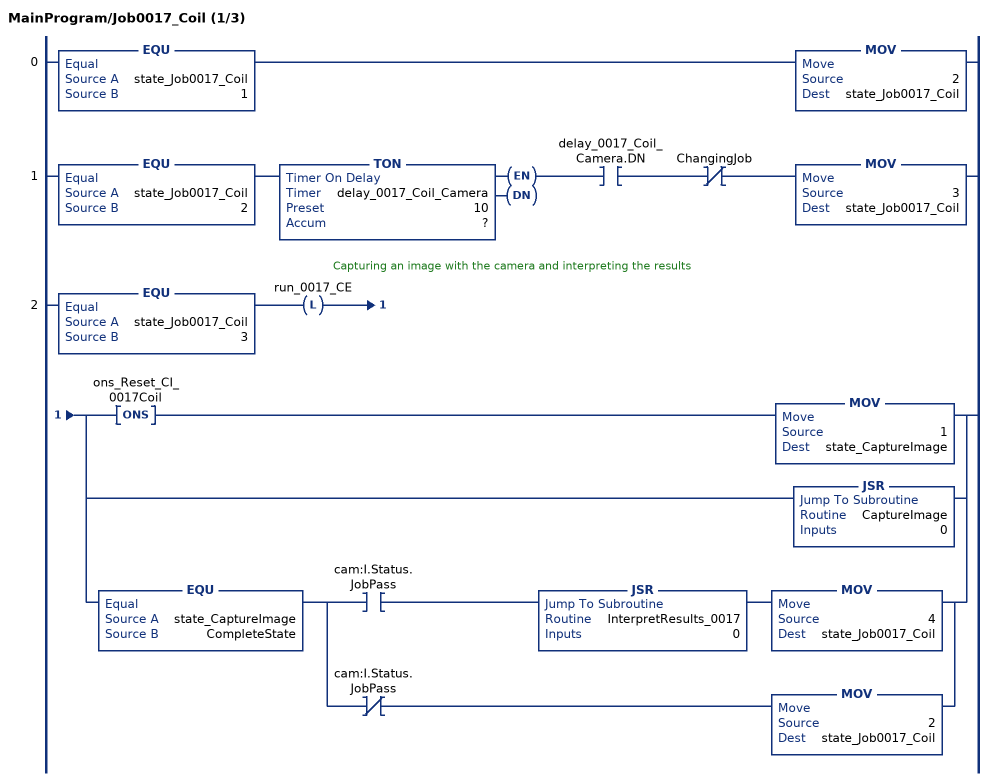
   0: EQU(state_Job0017_Coil,1)MOV(2,state_Job0017_Coil);
   1: EQU(state_Job0017_Coil,2)TON(delay_0017_Coil_Camera,?,?)XIC(delay_0017_Coil_Camera.DN)XIO(ChangingJob)MOV(3,state_Job0017_Coil);
   // Capturing an image with the camera and interpreting the results
   2: EQU(state_Job0017_Coil,3)OTL(run_0017_CE)[[ONS(ons_Reset_CI_0017Coil) MOV(1,state_CaptureImage) ,JSR(CaptureImage,0) ] ,EQU(state_CaptureImage,CompleteState) [XIC(cam:I.Status.JobPass) JSR(InterpretResults_0017,0) MOV(4,state_Job0017_Coil) ,XIO(cam:I.Status.JobPass) MOV(2,state_Job0017_Coil) ] ];
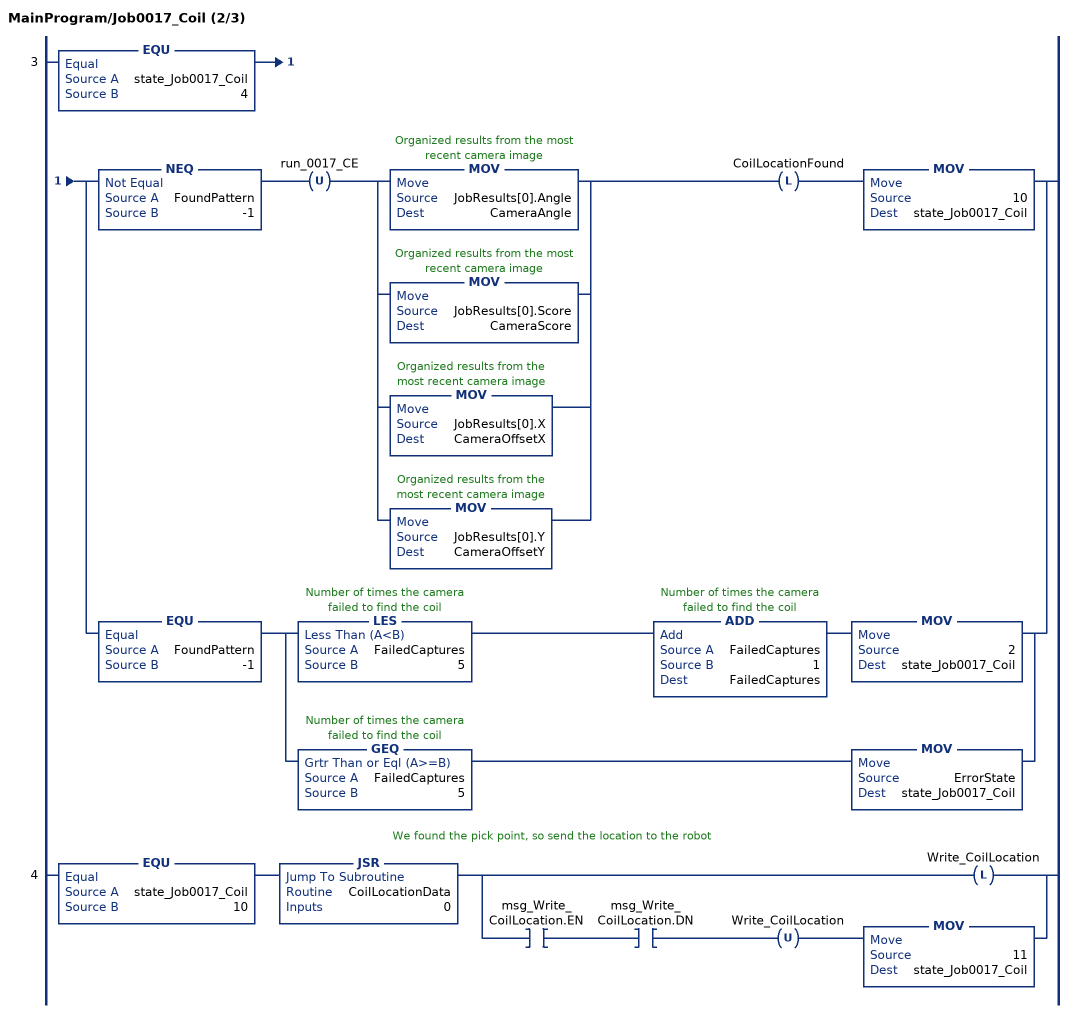
   3: EQU(state_Job0017_Coil,4)[NEQ(FoundPattern,-1) OTU(run_0017_CE) [MOV(JobResults[0].Angle,CameraAngle) ,MOV(JobResults[0].Score,CameraScore) ,MOV(JobResults[0].X,CameraOffsetX) ,MOV(JobResults[0].Y,CameraOffsetY) ] OTL(CoilLocationFound) MOV(10,state_Job0017_Coil) ,EQU(FoundPattern,-1) [LES(FailedCaptures,5) ADD(FailedCaptures,1,FailedCaptures) MOV(2,state_Job0017_Coil) ,GEQ(FailedCaptures,5) MOV(ErrorState,state_Job0017_Coil) ] ];
   // We found the pick point, so send the location to the robot
   4: EQU(state_Job0017_Coil,10)JSR(CoilLocationData,0)[OTL(Write_CoilLocation) ,XIC(msg_Write_CoilLocation.EN) XIC(msg_Write_CoilLocation.DN) OTU(Write_CoilLocation) MOV(11,state_Job0017_Coil) ];
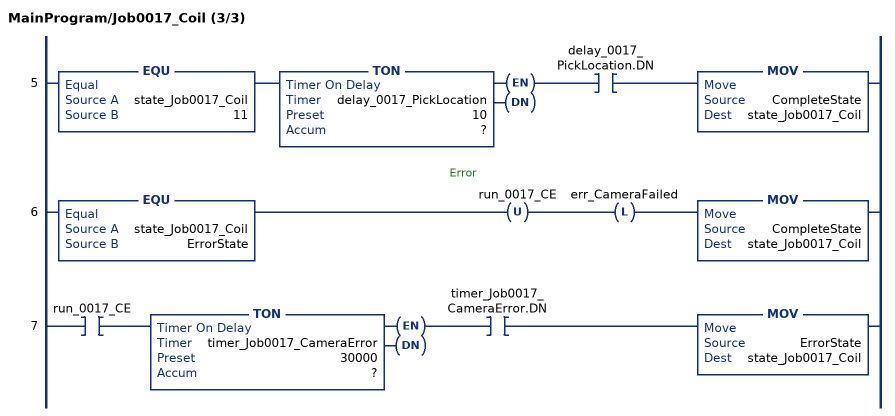
   5: EQU(state_Job0017_Coil,11)TON(delay_0017_PickLocation,?,?)XIC(delay_0017_PickLocation.DN)MOV(CompleteState,state_Job0017_Coil);
   // Error
   6: EQU(state_Job0017_Coil,ErrorState)OTU(run_0017_CE)OTL(err_CameraFailed)MOV(CompleteState,state_Job0017_Coil);
   7: XIC(run_0017_CE)TON(timer_Job0017_CameraError,?,?)XIC(timer_Job0017_CameraError.DN)MOV(ErrorState,state_Job0017_Coil);
END_ROUTINE

ROUTINE Job0017_Orient   (* ladder *)
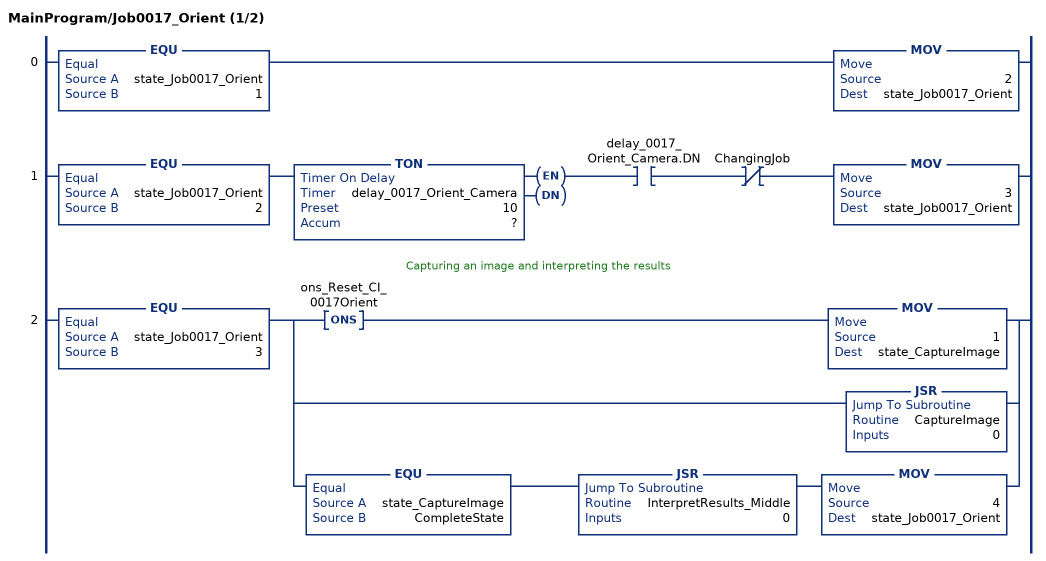
   0: EQU(state_Job0017_Orient,1)MOV(2,state_Job0017_Orient);
   1: EQU(state_Job0017_Orient,2)TON(delay_0017_Orient_Camera,?,?)XIC(delay_0017_Orient_Camera.DN)XIO(ChangingJob)MOV(3,state_Job0017_Orient);
   // Capturing an image and interpreting the results
   2: EQU(state_Job0017_Orient,3)[[ONS(ons_Reset_CI_0017Orient) MOV(1,state_CaptureImage) ,JSR(CaptureImage,0) ] ,EQU(state_CaptureImage,CompleteState) JSR(InterpretResults_Middle,0) MOV(4,state_Job0017_Orient) ];
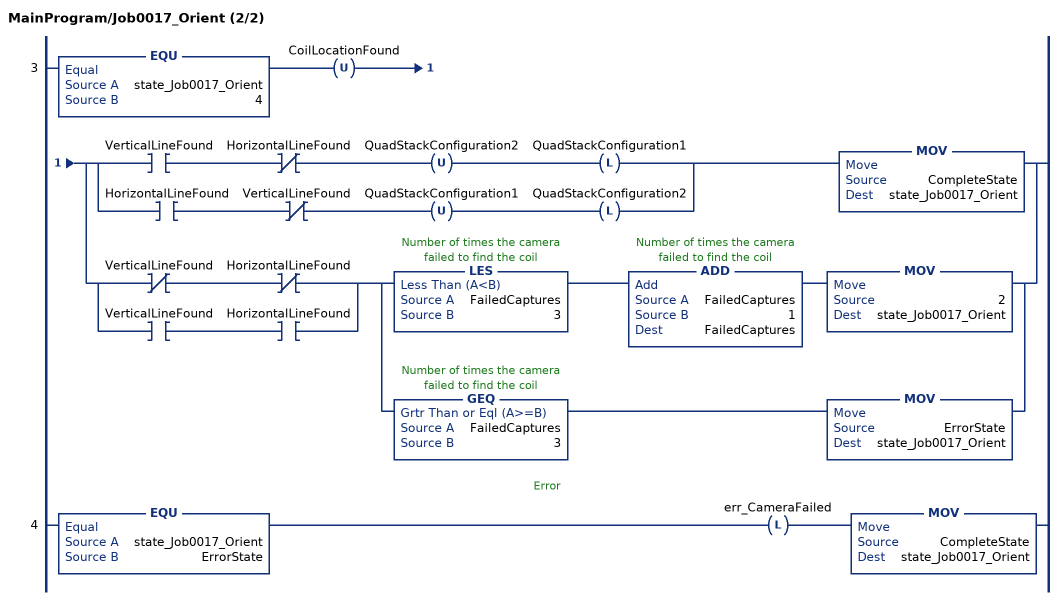
   3: EQU(state_Job0017_Orient,4)OTU(CoilLocationFound)[[XIC(VerticalLineFound) XIO(HorizontalLineFound) OTU(QuadStackConfiguration2) OTL(QuadStackConfiguration1) ,XIC(HorizontalLineFound) XIO(VerticalLineFound) OTU(QuadStackConfiguration1) OTL(QuadStackConfiguration2) ] MOV(CompleteState,state_Job0017_Orient) ,[XIO(VerticalLineFound) XIO(HorizontalLineFound) ,XIC(VerticalLineFound) XIC(HorizontalLineFound) ] [LES(FailedCaptures,3) ADD(FailedCaptures,1,FailedCaptures) MOV(2,state_Job0017_Orient) ,GEQ(FailedCaptures,3) MOV(ErrorState,state_Job0017_Orient) ] ];
   // Error
   4: EQU(state_Job0017_Orient,ErrorState)OTL(err_CameraFailed)MOV(CompleteState,state_Job0017_Orient);
END_ROUTINE

ROUTINE Job2832   (* ladder *)
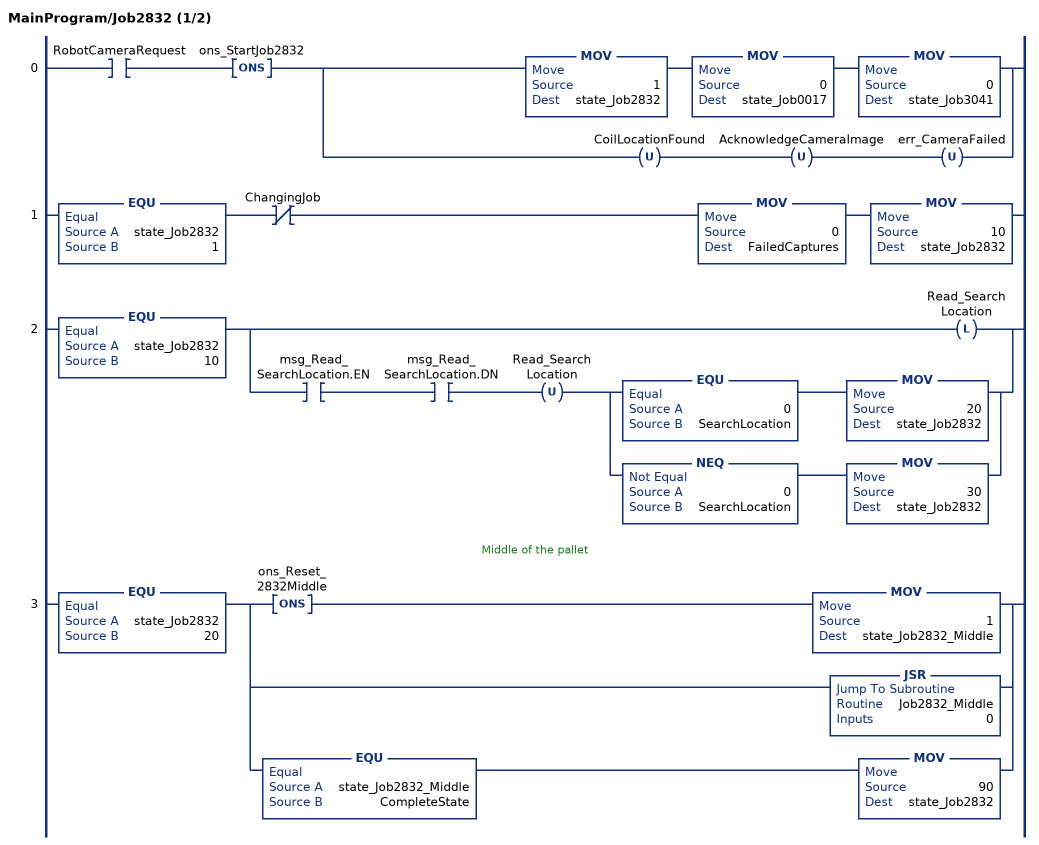
   0: XIC(RobotCameraRequest)ONS(ons_StartJob2832)[MOV(1,state_Job2832) MOV(0,state_Job0017) MOV(0,state_Job3041) ,OTU(CoilLocationFound) OTU(AcknowledgeCameraImage) OTU(err_CameraFailed) ];
   1: EQU(state_Job2832,1)XIO(ChangingJob)MOV(0,FailedCaptures)MOV(10,state_Job2832);
   2: EQU(state_Job2832,10)[OTL(Read_SearchLocation) ,XIC(msg_Read_SearchLocation.EN) XIC(msg_Read_SearchLocation.DN) OTU(Read_SearchLocation) [EQU(0,SearchLocation) MOV(20,state_Job2832) ,NEQ(0,SearchLocation) MOV(30,state_Job2832) ] ];
   // Middle of the pallet
   3: EQU(state_Job2832,20)[[ONS(ons_Reset_2832Middle) MOV(1,state_Job2832_Middle) ,JSR(Job2832_Middle,0) ] ,EQU(state_Job2832_Middle,CompleteState) MOV(90,state_Job2832) ];
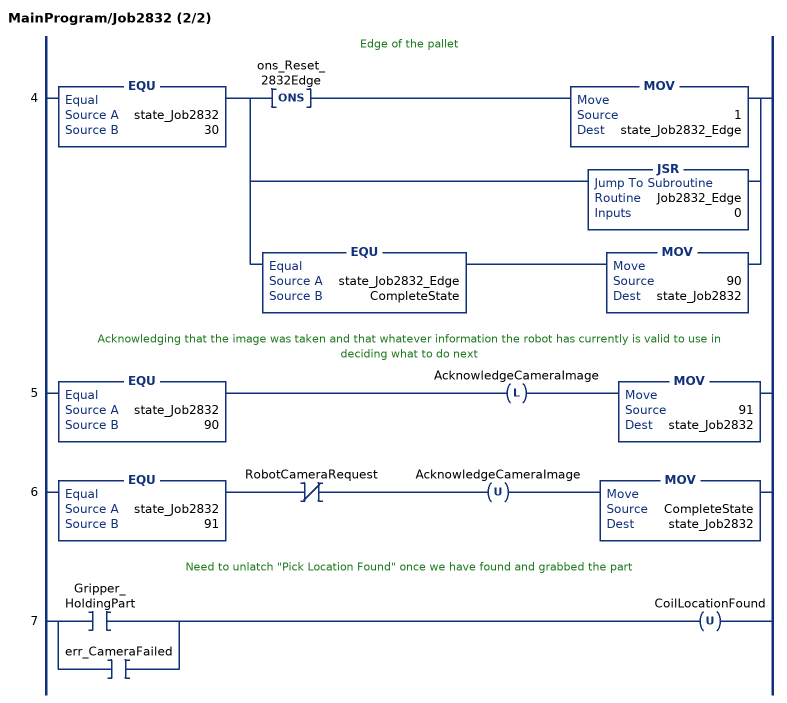
   // Edge of the pallet
   4: EQU(state_Job2832,30)[[ONS(ons_Reset_2832Edge) MOV(1,state_Job2832_Edge) ,JSR(Job2832_Edge,0) ] ,EQU(state_Job2832_Edge,CompleteState) MOV(90,state_Job2832) ];
   // Acknowledging that the image was taken and that whatever information the robot has currently is valid to use in deciding what to do next
   5: EQU(state_Job2832,90)OTL(AcknowledgeCameraImage)MOV(91,state_Job2832);
   6: EQU(state_Job2832,91)XIO(RobotCameraRequest)OTU(AcknowledgeCameraImage)MOV(CompleteState,state_Job2832);
   // Need to unlatch "Pick Location Found" once we have found and grabbed the part
   7: [XIC(Gripper_HoldingPart) ,XIC(err_CameraFailed) ]OTU(CoilLocationFound);
END_ROUTINE
